// SIMATIC S7-200 project (STEP 7-Micro/WIN), CPU 224 AM REL 21.02

SYMBOL_TABLE 用户定义1
对应40100地址        VW1198
对应40001地址        VW1000
对应30016地址        AIW30
END_SYMBOL_TABLE

SYMBOL_TABLE S7-200 符号
Always_On        SM0.0    // 始终接通为 ON
First_Scan_On    SM0.1    // 仅第一个扫描周期中接通为 ON
END_SYMBOL_TABLE

ORGANIZATION_BLOCK 主程序:OB1
TITLE=程序注释
BEGIN
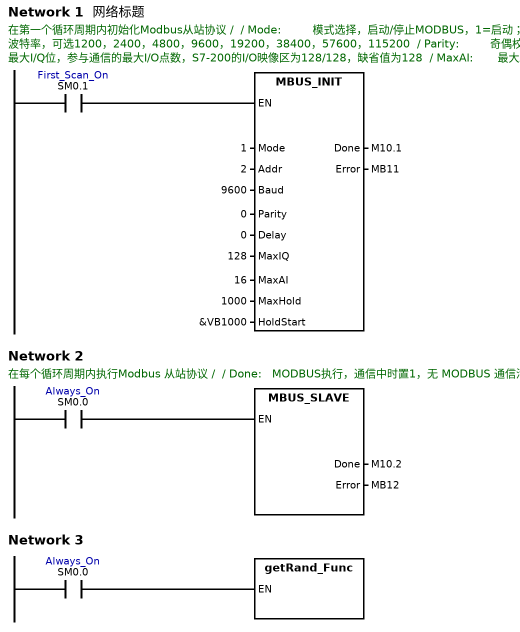
Network 1 // 网络标题
// 在第一个循环周期内初始化Modbus从站协议
// 
// Mode:         模式选择，启动/停止MODBUS，1=启动；0=停止
// Address:     从站地址，MODBUS从站地址，取值1~247
// Baud:         波特率，可选1200，2400，4800，9600，19200，38400，57600，115200 
// Parity:         奇偶校验，0=无校验；1=奇校验；2=偶校验 
// Delay:         延时，附加字符间延时，缺省值为0 
// MaxIQ:       最大I/Q位，参与通信的最大I/O点数，S7-200的I/O映像区为128/128，缺省值为128 
// MaxAI:       最大AI字数，参与通信的最大AI通道数，可为16或32 
// MaxHold:   最大保持寄存器区，参与通信的V存储区字（VW） 
// HoldStart:   保持寄存器区起始地址，以&VBx指定（间接寻址方式） 
// 
// Done:        初始化完成标志，成功初始化后置1 
// Error:         初始化错误代码
// 
// 在本例子中，设置从站地址为1
// Port0 通讯波特率为9600
// 无校验
// 可以使用的S7-200最大数字量输入输出点数为128
// 可以使用的S7-200最大模拟量输入寄存器字数为32
// 可以使用的V区寄存器地址字数为100（最大可填一千多个字都没问题）， 起始地址为VB1000
// 
// 注意：本例子中，Modbus RTU 从站指令使用的库存储为VB0---VB779，这段寄存器地址不能再被程序中的任何指令使用，包括MBUS_INIT 和 MBUS_SLAVE 指令在内
LD     First_Scan_On:SM0.1
CALL   MBUS_INIT:SBR3, 1, 2, 9600, 0, 0, 128, 16, 1000, &VB1000, M10.1, MB11
Network 2
// 在每个循环周期内执行Modbus 从站协议
// 
// Done:   MODBUS执行，通信中时置1，无 MODBUS 通信活动时为 0
// Error:    错误代码：0=无错误 
LD     Always_On:SM0.0
CALL   MBUS_SLAVE:SBR1, M10.2, MB12
Network 3
LD     Always_On:SM0.0
CALL   getRand_Func:SBR4
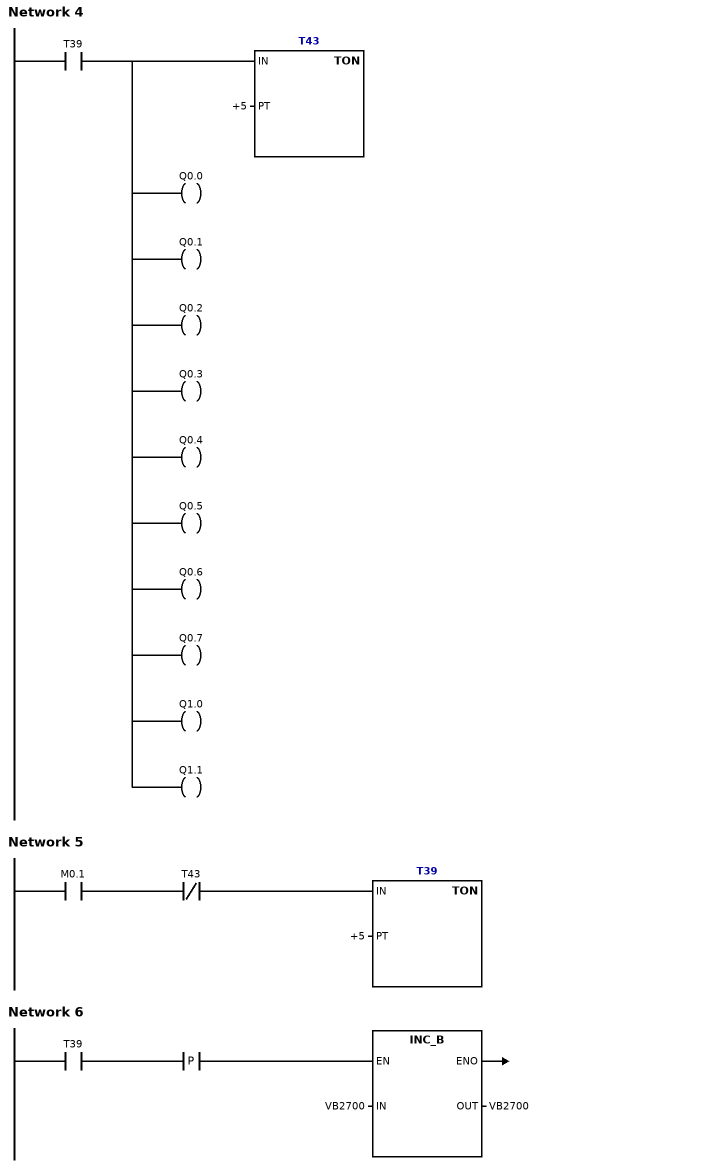
Network 4
LD     T39
TON    T43, +5
=      Q0.0
=      Q0.1
=      Q0.2
=      Q0.3
=      Q0.4
=      Q0.5
=      Q0.6
=      Q0.7
=      Q1.0
=      Q1.1
Network 5
LD     M0.1
AN     T43
TON    T39, +5
Network 6
LD     T39
EU
INCB   VB2700
END_ORGANIZATION_BLOCK

// SBR1: protected block, not included

// SBR2: protected block, not included

// SBR3: protected block, not included

SUBROUTINE_BLOCK getRand_Func:SBR4
TITLE=
BEGIN
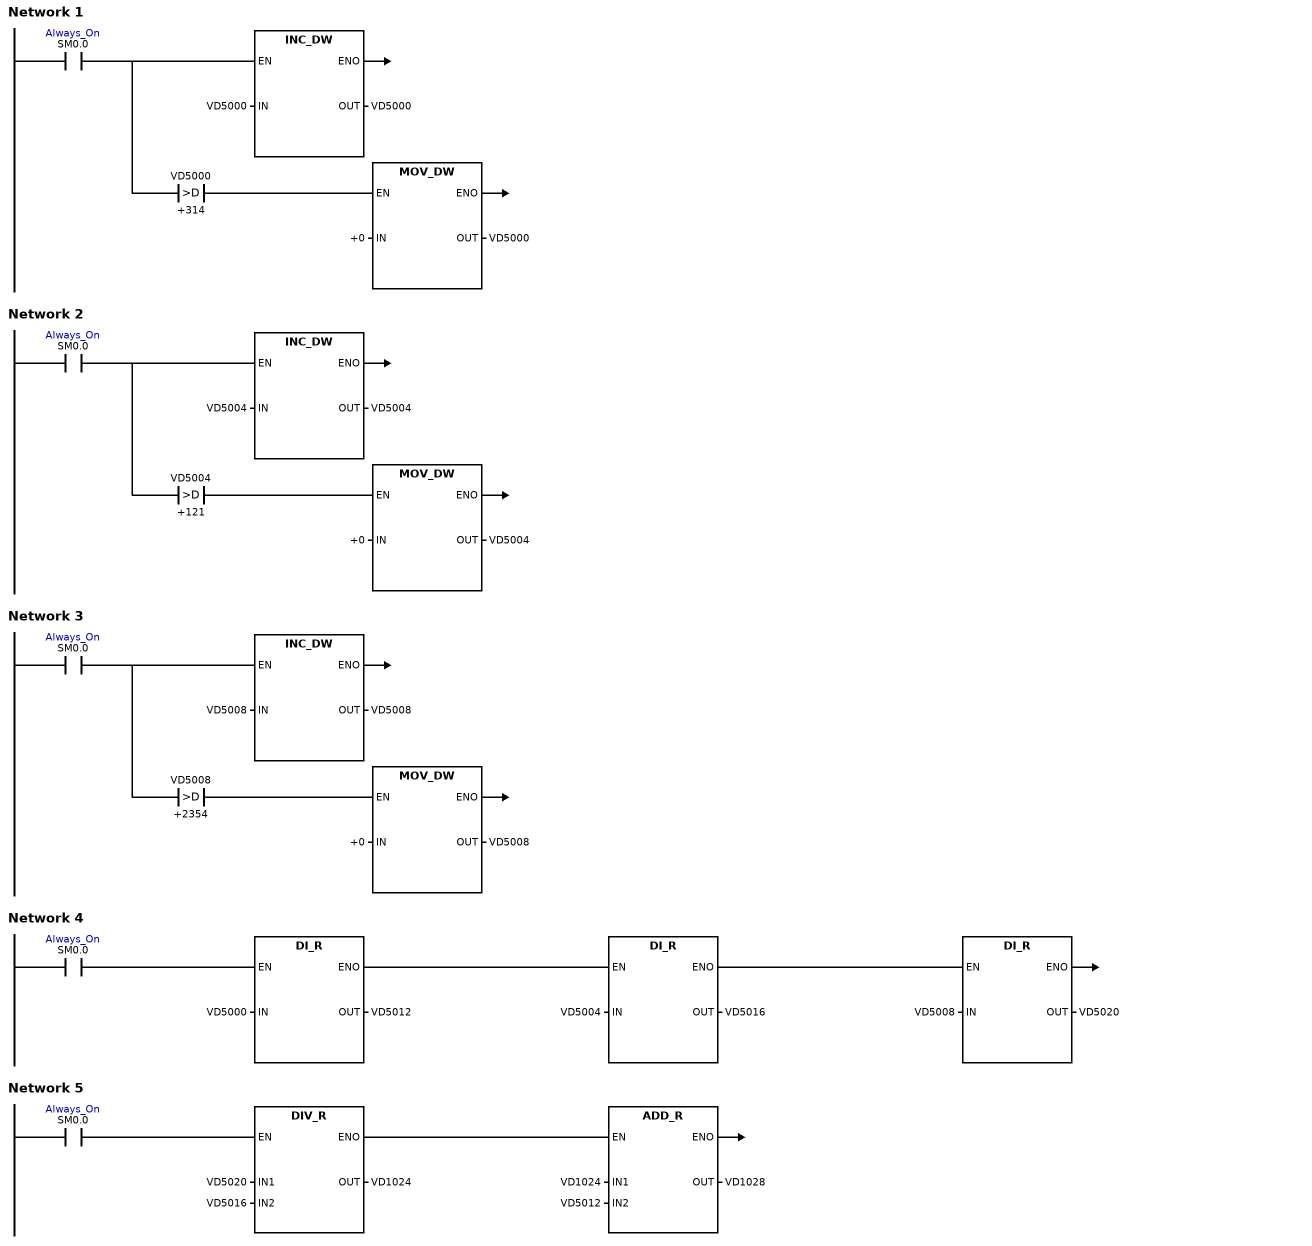
Network 1
LD     Always_On:SM0.0
INCD   VD5000
AD>    VD5000, +314
MOVD   +0, VD5000
Network 2
LD     Always_On:SM0.0
INCD   VD5004
AD>    VD5004, +121
MOVD   +0, VD5004
Network 3
LD     Always_On:SM0.0
INCD   VD5008
AD>    VD5008, +2354
MOVD   +0, VD5008
Network 4
LD     Always_On:SM0.0
DTR    VD5000, VD5012
AENO
DTR    VD5004, VD5016
AENO
DTR    VD5008, VD5020
Network 5
LD     Always_On:SM0.0
MOVR   VD5020, VD1024
AENO
/R     VD5016, VD1024
AENO
MOVR   VD1024, VD1028
+R     VD5012, VD1028
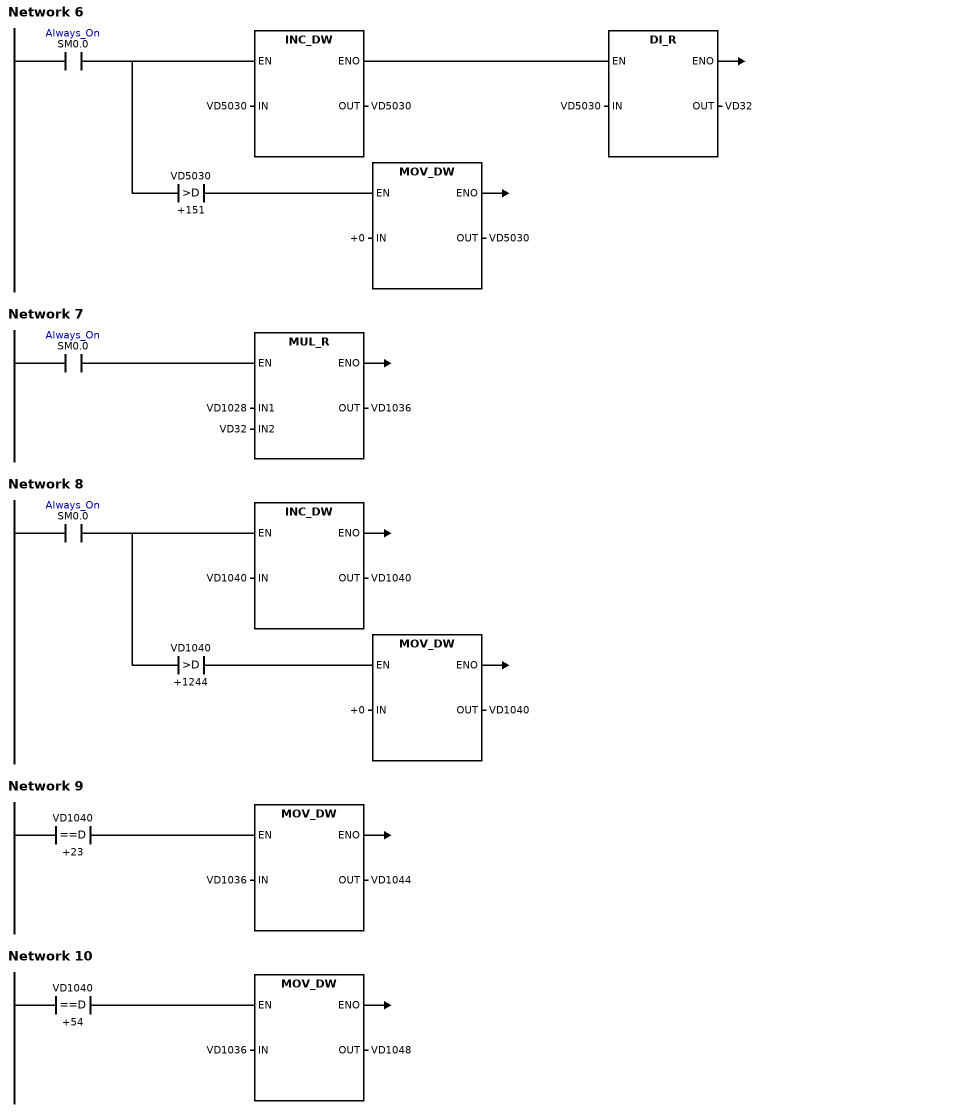
Network 6
LD     Always_On:SM0.0
LPS
INCD   VD5030
AENO
DTR    VD5030, VD32
LPP
AD>    VD5030, +151
MOVD   +0, VD5030
Network 7
LD     Always_On:SM0.0
MOVR   VD1028, VD1036
*R     VD32, VD1036
Network 8
LD     Always_On:SM0.0
INCD   VD1040
AD>    VD1040, +1244
MOVD   +0, VD1040
Network 9
LDD=   VD1040, +23
MOVD   VD1036, VD1044
Network 10
LDD=   VD1040, +54
MOVD   VD1036, VD1048
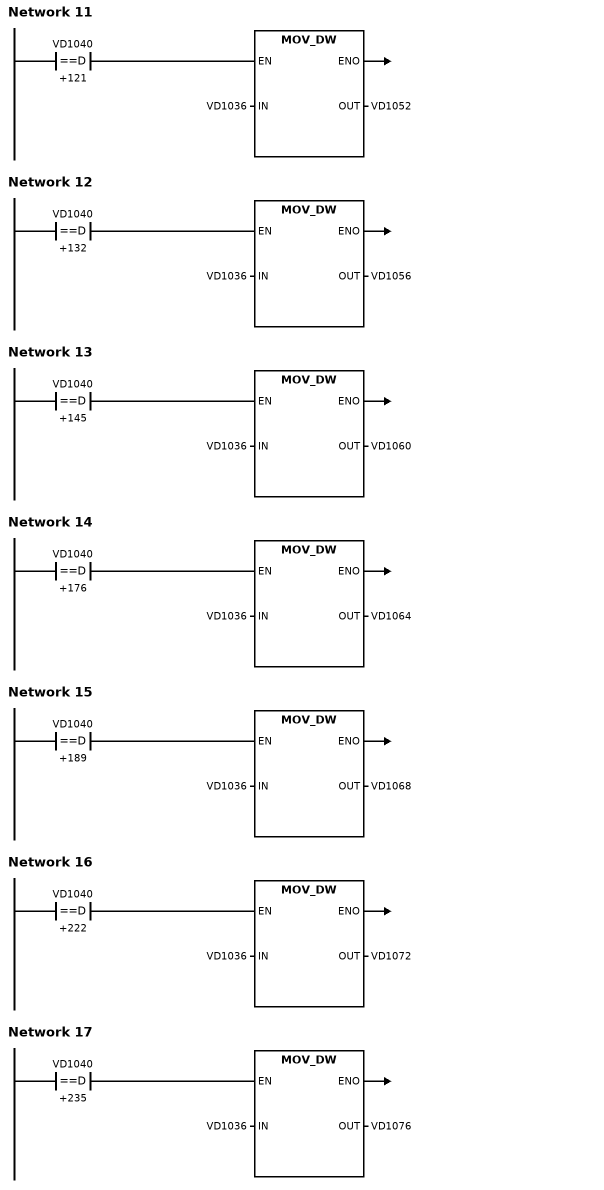
Network 11
LDD=   VD1040, +121
MOVD   VD1036, VD1052
Network 12
LDD=   VD1040, +132
MOVD   VD1036, VD1056
Network 13
LDD=   VD1040, +145
MOVD   VD1036, VD1060
Network 14
LDD=   VD1040, +176
MOVD   VD1036, VD1064
Network 15
LDD=   VD1040, +189
MOVD   VD1036, VD1068
Network 16
LDD=   VD1040, +222
MOVD   VD1036, VD1072
Network 17
LDD=   VD1040, +235
MOVD   VD1036, VD1076
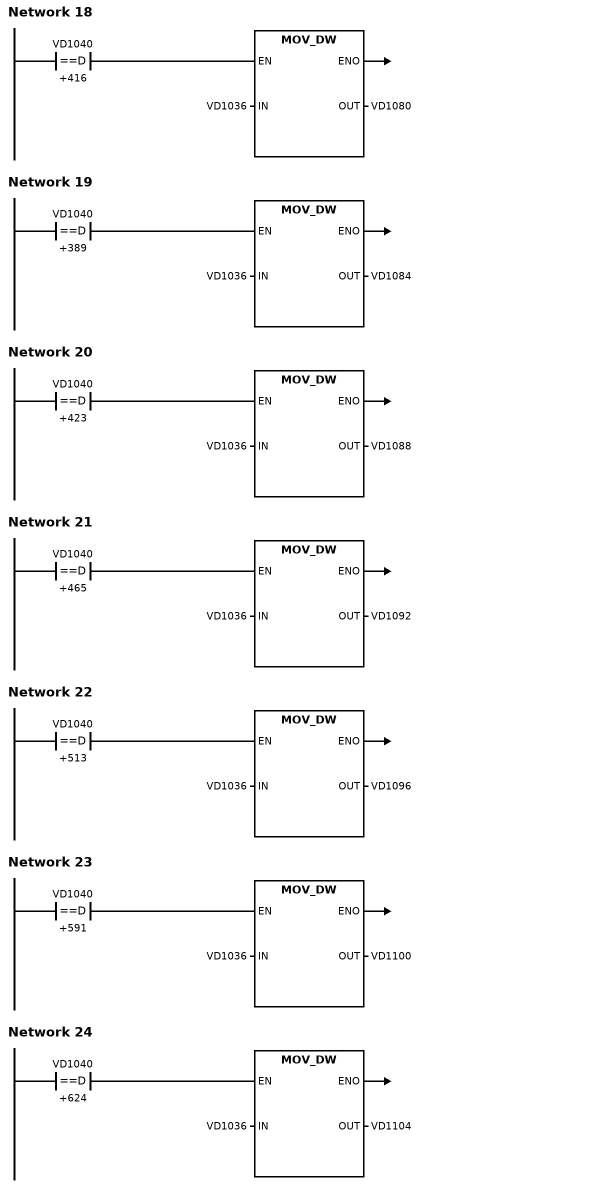
Network 18
LDD=   VD1040, +416
MOVD   VD1036, VD1080
Network 19
LDD=   VD1040, +389
MOVD   VD1036, VD1084
Network 20
LDD=   VD1040, +423
MOVD   VD1036, VD1088
Network 21
LDD=   VD1040, +465
MOVD   VD1036, VD1092
Network 22
LDD=   VD1040, +513
MOVD   VD1036, VD1096
Network 23
LDD=   VD1040, +591
MOVD   VD1036, VD1100
Network 24
LDD=   VD1040, +624
MOVD   VD1036, VD1104
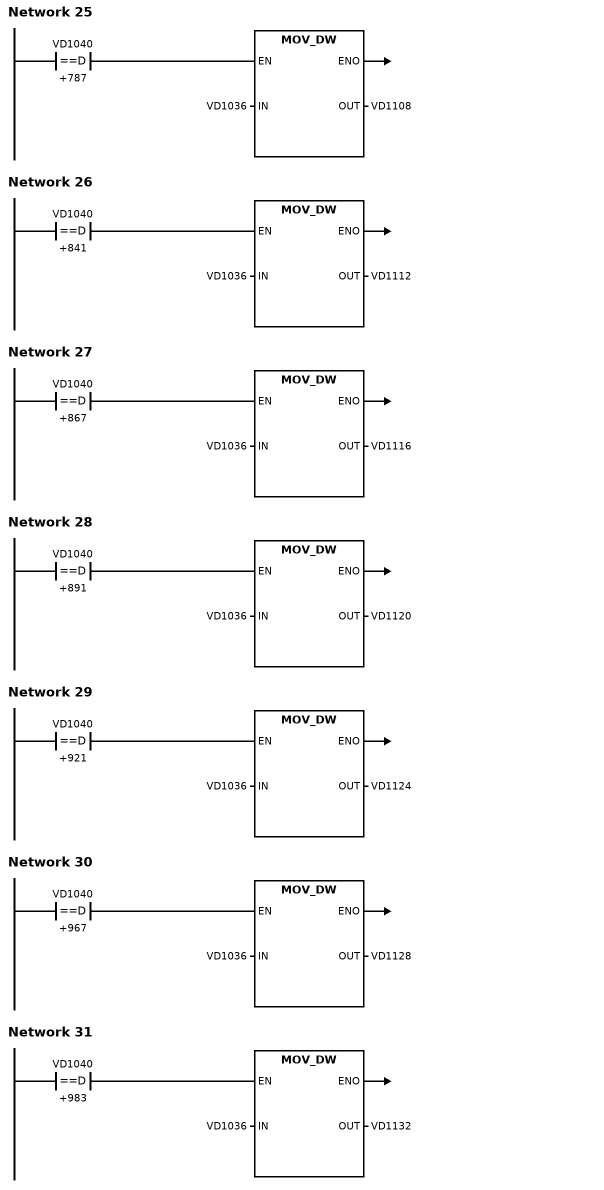
Network 25
LDD=   VD1040, +787
MOVD   VD1036, VD1108
Network 26
LDD=   VD1040, +841
MOVD   VD1036, VD1112
Network 27
LDD=   VD1040, +867
MOVD   VD1036, VD1116
Network 28
LDD=   VD1040, +891
MOVD   VD1036, VD1120
Network 29
LDD=   VD1040, +921
MOVD   VD1036, VD1124
Network 30
LDD=   VD1040, +967
MOVD   VD1036, VD1128
Network 31
LDD=   VD1040, +983
MOVD   VD1036, VD1132
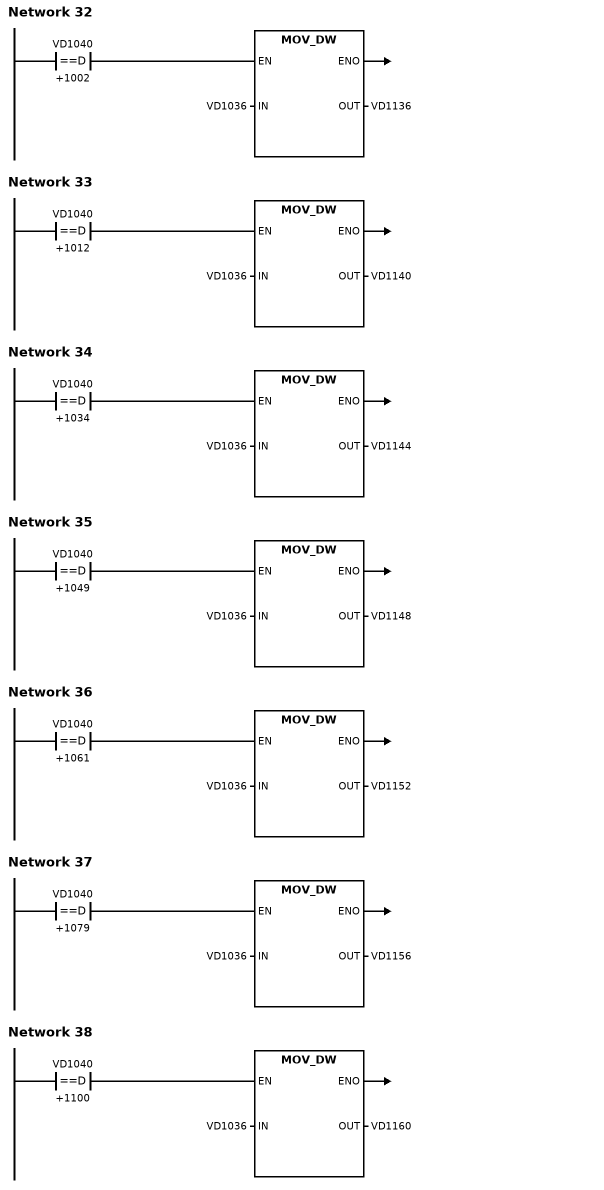
Network 32
LDD=   VD1040, +1002
MOVD   VD1036, VD1136
Network 33
LDD=   VD1040, +1012
MOVD   VD1036, VD1140
Network 34
LDD=   VD1040, +1034
MOVD   VD1036, VD1144
Network 35
LDD=   VD1040, +1049
MOVD   VD1036, VD1148
Network 36
LDD=   VD1040, +1061
MOVD   VD1036, VD1152
Network 37
LDD=   VD1040, +1079
MOVD   VD1036, VD1156
Network 38
LDD=   VD1040, +1100
MOVD   VD1036, VD1160
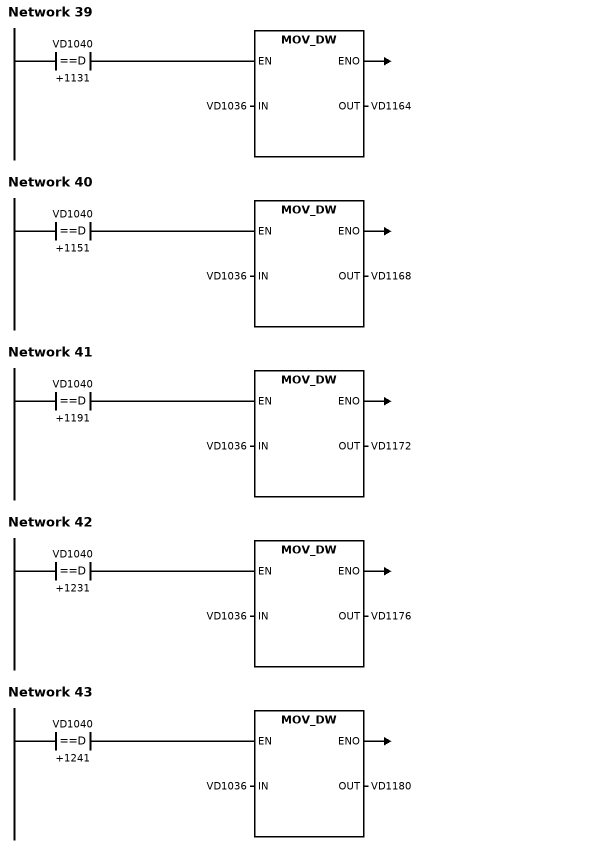
Network 39
LDD=   VD1040, +1131
MOVD   VD1036, VD1164
Network 40
LDD=   VD1040, +1151
MOVD   VD1036, VD1168
Network 41
LDD=   VD1040, +1191
MOVD   VD1036, VD1172
Network 42
LDD=   VD1040, +1231
MOVD   VD1036, VD1176
Network 43
LDD=   VD1040, +1241
MOVD   VD1036, VD1180
Network 45 // Network Title
// Network Comment
END_SUBROUTINE_BLOCK
